FUNCTION "FC_SPL_PLC1" : VOID
TITLE =
//$Revision: 1.12 $
//$Date: 2007/10/19 12:45:04CEST $
//$Author: hgc $
//
//
//
//PLC-SPL Baustein für Solutionline DMx55-125x2
//
//Unterteilt in zwei Sicherheitsbereiche:
//1. Bereich 1         (Arbeitsraumachsen / Palettenwechslerachse / Mgazinachsen)
//bestehend aus Achse:    X Y Z B C SPI              PW             MAG1/MAG2 GR
//
//2. Bereich 2         (Palettenspeicherachsen / Palettenwechslerachse)
//bestehend aus Achse:     DREHST/TRANSP/HUB              PW
//
AUTHOR : GehAB
FAMILY : SPL
VERSION : 3.0


VAR_TEMP
  TX_ABNAHME_TEST_SBH_AKT : BOOL ;
END_VAR
BEGIN
NETWORK
TITLE =PLC-->NC: Vorbesetzungen
// Reissleine
      SET   ;
      =     "DB_SPL".IPLC_NEG_NOT_HALT;
      =     "DB_SIEM_NCK".A_Disabl_Out1;
      =     "DB_SIEM_NCK".A_OvMask_Out1;
      =     "DB_SIEM_NCK".A_Set_Out1;
      CLR   ;
      =     "DB_SIEM_NCK".A_Disabl_Out2;
      =     "DB_SIEM_NCK".A_Disabl_Out3;
      SET   ;
      =     "DB_SIEM_NCK".A_OvMask_Out2;
      =     "DB_SIEM_NCK".A_OvMask_Out3;
NETWORK
TITLE =PLC-->NC: Safety Abnahme läuft
// kein NOT-AUS auslösen und nicht SBH/SG abwählen bei Fehler SG/SGH
      U     "DB_PLC_MD_DB20".UDHex._05_BIT2_SAFTY_ABNAHME;
      =     "DB_SPL".IPLC_Abnahme;
NETWORK
TITLE =PLC-->NC: Zwangsdynamisierung laeuft
//kein Not-AUS auslösen
      U(    ;
      U(    ;
      O     "DB_SAFE_ZD".Seco_Test.Test_HW_laueft;
      O     "DB_SAFE_ZD".Seco_Test.Test_ABSP_laeuft;
      O     "DB_SAFE_ZD".Seco_Test.Test_extStop_laeuft;
      O     "DB_SAFE_ZD".Seco_Test.Test_Bremse_laeuft;
      O     ;
      U(    ;
      O     "DB_SAFE_ZD".Seco_Test.BER2_Test_HW_laueft;
      O     "DB_SAFE_ZD".Seco_Test.BER2_Test_ABSP_laeuft;
      O     "DB_SAFE_ZD".Seco_Test.BER2_Test_extStop_laeuft;
      O     "DB_SAFE_ZD".Seco_Test.BER2_Test_Bremse_laeuft;
      )     ;
      UN    "m_inbetrieb_logisch_1";
      )     ;
      S     "DB_SAFE_ALLG1".M_IMP_Test_HW_laueft;
      U(    ;
      U(    ;
      O     "DB_SAFE_ZD".Seco_Test.Test_extStop_laeuft;
      O     ;
      U     "DB_SAFE_ZD".Seco_Test.BER2_Test_extStop_laeuft;
      UN    "m_inbetrieb_logisch_1";
      )     ;
      FN    "DB_SAFE_ALLG1".M_FP_Test_HW_laueft;
      O     "M_Ruecksetze_Fehler";
      )     ;
      R     "DB_SAFE_ALLG1".M_IMP_Test_HW_laueft;
      U     "DB_SAFE_ALLG1".M_IMP_Test_HW_laueft;
      )     ;
      L     S5T#1S;
      SA    "T_SA_HW_Test_laeuft";
      NOP   0;
      NOP   0;
      NOP   0;
      U     "T_SA_HW_Test_laeuft";
      =     "DB_SPL".IPLC_ZD_GR1_RUN;
NETWORK
TITLE =PLC-->NC: ARBEITSRAUM: SBH Anforderung durch Anwahl Entriegeln
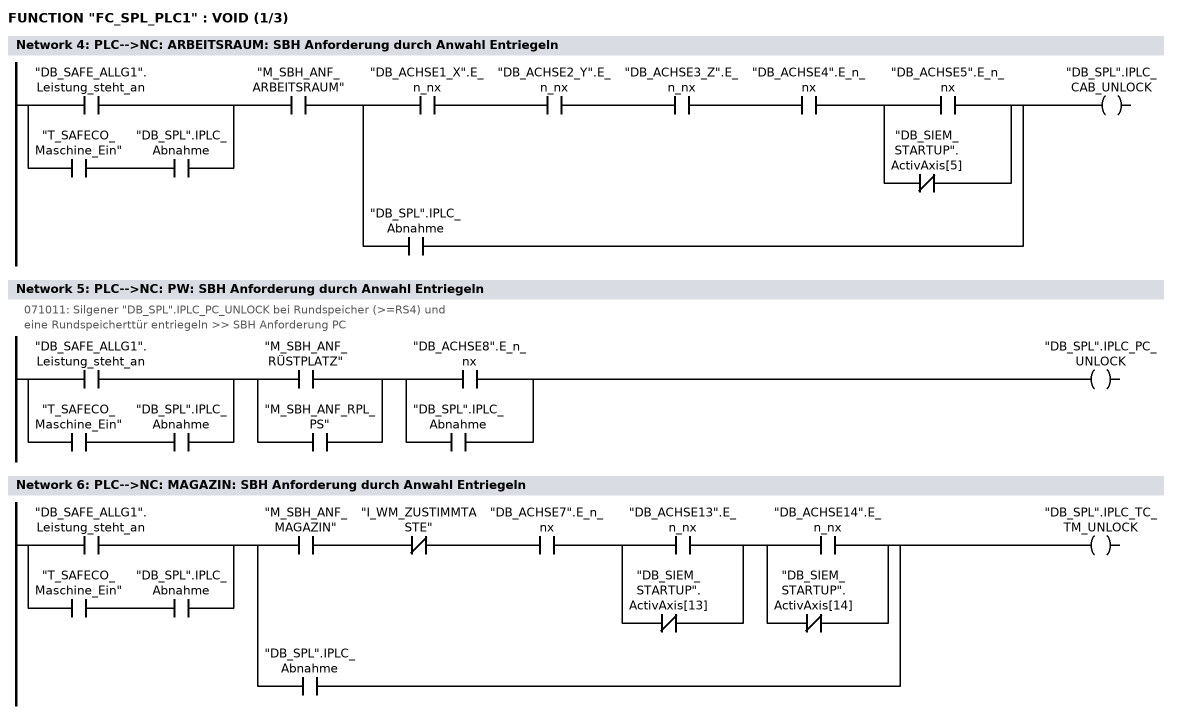

      U(    ;
      O     "DB_SAFE_ALLG1".Leistung_steht_an;
      O     ;
      U     "T_SAFECO_Maschine_Ein";
      U     "DB_SPL".IPLC_Abnahme;
      )     ;
      U     "M_SBH_ANF_ARBEITSRAUM";
      U(    ;
      U     "DB_ACHSE1_X".E_n_nx;
      U     "DB_ACHSE2_Y".E_n_nx;
      U     "DB_ACHSE3_Z".E_n_nx;
      U     "DB_ACHSE4".E_n_nx;
      U(    ;
      O     "DB_ACHSE5".E_n_nx;
      ON    "DB_SIEM_STARTUP".ActivAxis[5];
      )     ;
      O     "DB_SPL".IPLC_Abnahme;
      )     ;
      =     "DB_SPL".IPLC_CAB_UNLOCK;
NETWORK
TITLE =PLC-->NC: PW: SBH Anforderung durch Anwahl Entriegeln
//071011: Silgener "DB_SPL".IPLC_PC_UNLOCK bei Rundspeicher (>=RS4) und
//eine Rundspeicherttür entriegeln >> SBH Anforderung PC
      U(    ;
      O     "DB_SAFE_ALLG1".Leistung_steht_an;
      O     ;
      U     "T_SAFECO_Maschine_Ein";
      U     "DB_SPL".IPLC_Abnahme;
      )     ;
      U(    ;
      O     "M_SBH_ANF_RÜSTPLATZ";
      O     "M_SBH_ANF_RPL_PS";
      )     ;
      U(    ;
      O     "DB_ACHSE8".E_n_nx;
      O     "DB_SPL".IPLC_Abnahme;
      )     ;
      =     "DB_SPL".IPLC_PC_UNLOCK;
NETWORK
TITLE =PLC-->NC: MAGAZIN: SBH Anforderung durch Anwahl Entriegeln

      U(    ;
      O     "DB_SAFE_ALLG1".Leistung_steht_an;
      O     ;
      U     "T_SAFECO_Maschine_Ein";
      U     "DB_SPL".IPLC_Abnahme;
      )     ;
      U(    ;
      U     "M_SBH_ANF_MAGAZIN";
      UN    "I_WM_ZUSTIMMTASTE";
      U     "DB_ACHSE7".E_n_nx;
      U(    ;
      O     "DB_ACHSE13".E_n_nx;
      ON    "DB_SIEM_STARTUP".ActivAxis[13];
      )     ;
      U(    ;
      O     "DB_ACHSE14".E_n_nx;
      ON    "DB_SIEM_STARTUP".ActivAxis[14];
      )     ;
      O     "DB_SPL".IPLC_Abnahme;
      )     ;
      =     "DB_SPL".IPLC_TC_TM_UNLOCK;

NETWORK
TITLE =Sichere Eingänge auf Merker abbilden
//"DB_SPL".ISX_TM_DRIVES_EN_CNC  entspricht dem Eingang "IX_TC_ENABLE" (beide
//Signale durch PNOZ Multi gleichgeschaltet)
//
//"DB_SPL".ISX_PC_DRIVES_EN_CNC entspricht dem Eingang "IX_PC_ENABLE" (beide
//Signale durch PNOZ Multi gleichgeschaltet)
//
//Die Eingänge "IX_TC_ENABLE" und "IX_PC_ENABLE" werden im Rangierer auf
//Dummymerker gelegt. In der PLC wird nur das Profisafeeingangssignal abgefragt.
//
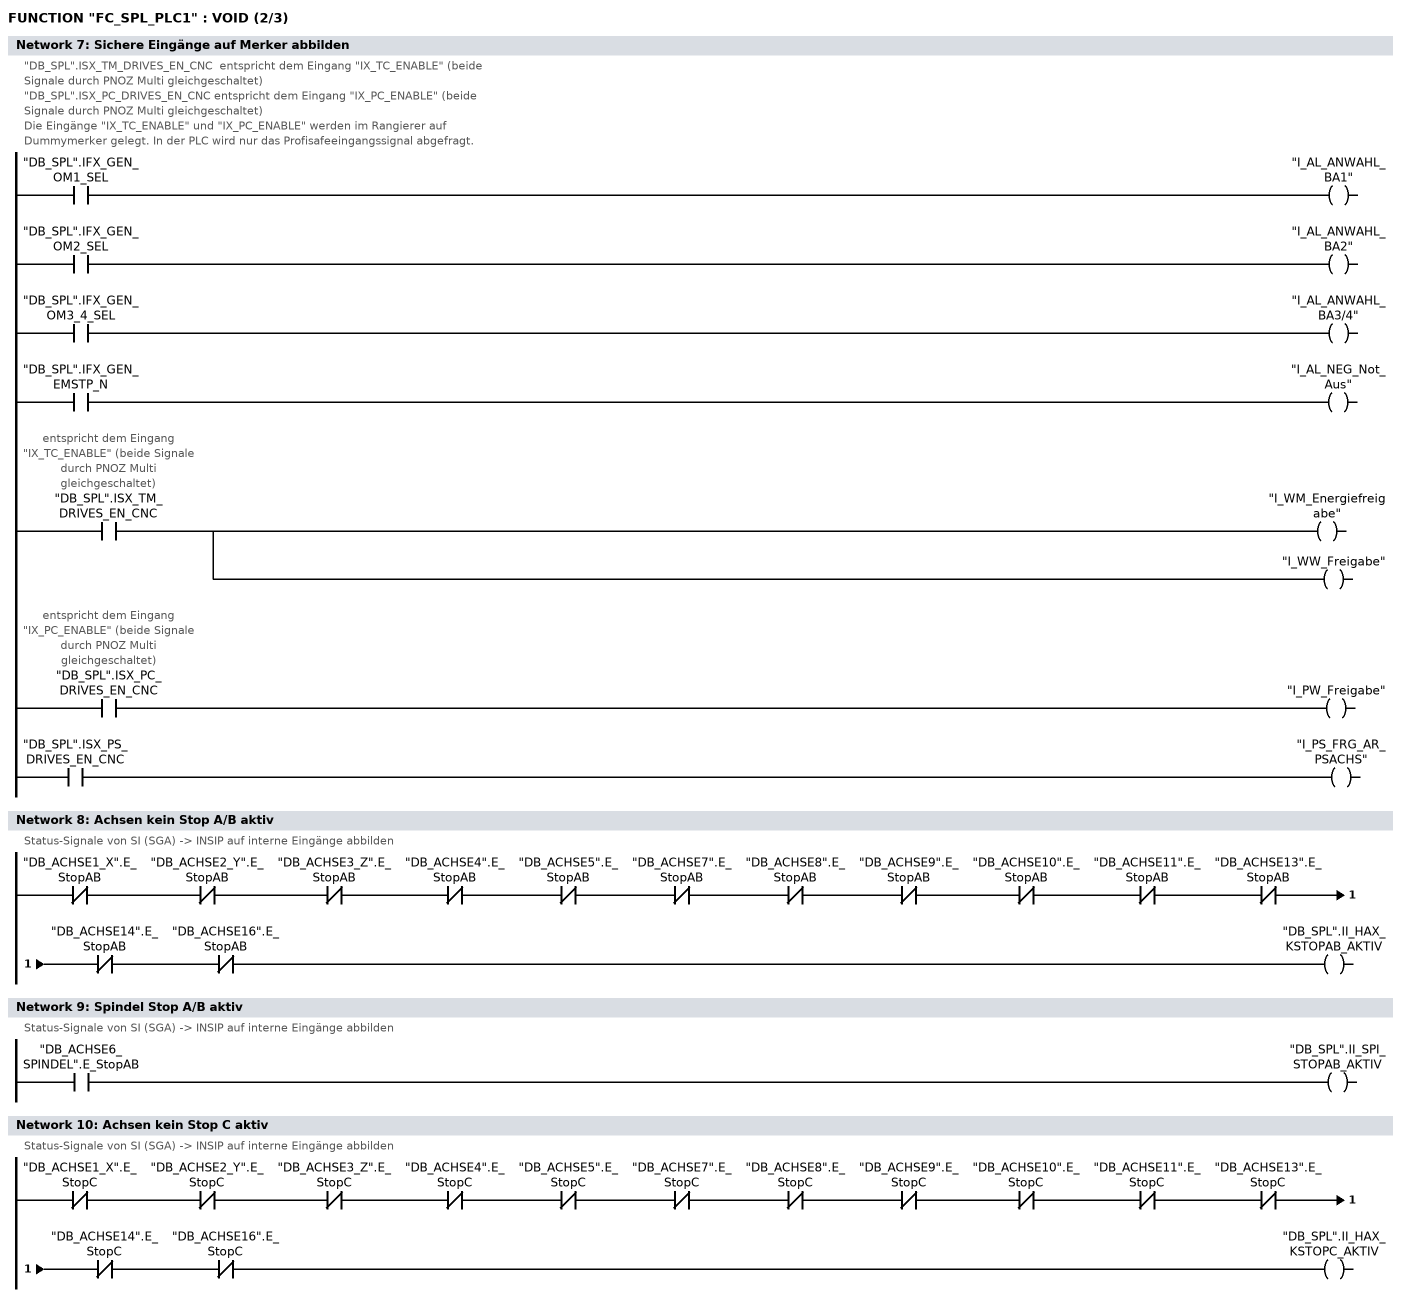
      U     "DB_SPL".IFX_GEN_OM1_SEL;
      =     "I_AL_ANWAHL_BA1";

      U     "DB_SPL".IFX_GEN_OM2_SEL;
      =     "I_AL_ANWAHL_BA2";

      U     "DB_SPL".IFX_GEN_OM3_4_SEL;
      =     "I_AL_ANWAHL_BA3/4";

      U     "DB_SPL".IFX_GEN_EMSTP_N;
      =     "I_AL_NEG_Not_Aus";

      U     "DB_SPL".ISX_TM_DRIVES_EN_CNC; // entspricht dem Eingang "IX_TC_ENABLE" (beide Signale durch PNOZ Multi gleichgeschaltet)
      =     "I_WM_Energiefreigabe";
      =     "I_WW_Freigabe";

      U     "DB_SPL".ISX_PC_DRIVES_EN_CNC; // entspricht dem Eingang "IX_PC_ENABLE" (beide Signale durch PNOZ Multi gleichgeschaltet)
      =     "I_PW_Freigabe";

      U     "DB_SPL".ISX_PS_DRIVES_EN_CNC;
      =     "I_PS_FRG_AR_PSACHS";
NETWORK
TITLE =Achsen kein Stop A/B aktiv
//Status-Signale von SI (SGA) -> INSIP auf interne Eingänge abbilden
      UN    "DB_ACHSE1_X".E_StopAB;
      UN    "DB_ACHSE2_Y".E_StopAB;
      UN    "DB_ACHSE3_Z".E_StopAB;
      UN    "DB_ACHSE4".E_StopAB;
      UN    "DB_ACHSE5".E_StopAB;
      UN    "DB_ACHSE7".E_StopAB;
      UN    "DB_ACHSE8".E_StopAB;
      UN    "DB_ACHSE9".E_StopAB;
      UN    "DB_ACHSE10".E_StopAB;
      UN    "DB_ACHSE11".E_StopAB;
      UN    "DB_ACHSE13".E_StopAB;
      UN    "DB_ACHSE14".E_StopAB;
      UN    "DB_ACHSE16".E_StopAB;
      =     "DB_SPL".II_HAX_KSTOPAB_AKTIV;
NETWORK
TITLE =Spindel Stop A/B aktiv
//Status-Signale von SI (SGA) -> INSIP auf interne Eingänge abbilden
      U     "DB_ACHSE6_SPINDEL".E_StopAB;
      =     "DB_SPL".II_SPI_STOPAB_AKTIV;
NETWORK
TITLE =Achsen kein Stop C aktiv
//Status-Signale von SI (SGA) -> INSIP auf interne Eingänge abbilden
      UN    "DB_ACHSE1_X".E_StopC;
      UN    "DB_ACHSE2_Y".E_StopC;
      UN    "DB_ACHSE3_Z".E_StopC;
      UN    "DB_ACHSE4".E_StopC;
      UN    "DB_ACHSE5".E_StopC;
      UN    "DB_ACHSE7".E_StopC;
      UN    "DB_ACHSE8".E_StopC;
      UN    "DB_ACHSE9".E_StopC;
      UN    "DB_ACHSE10".E_StopC;
      UN    "DB_ACHSE11".E_StopC;
      UN    "DB_ACHSE13".E_StopC;
      UN    "DB_ACHSE14".E_StopC;
      UN    "DB_ACHSE16".E_StopC;
      =     "DB_SPL".II_HAX_KSTOPC_AKTIV;
NETWORK
TITLE =Spindel Stop C aktiv
//Status-Signale von SI (SGA) -> INSIP auf interne Eingänge abbilden
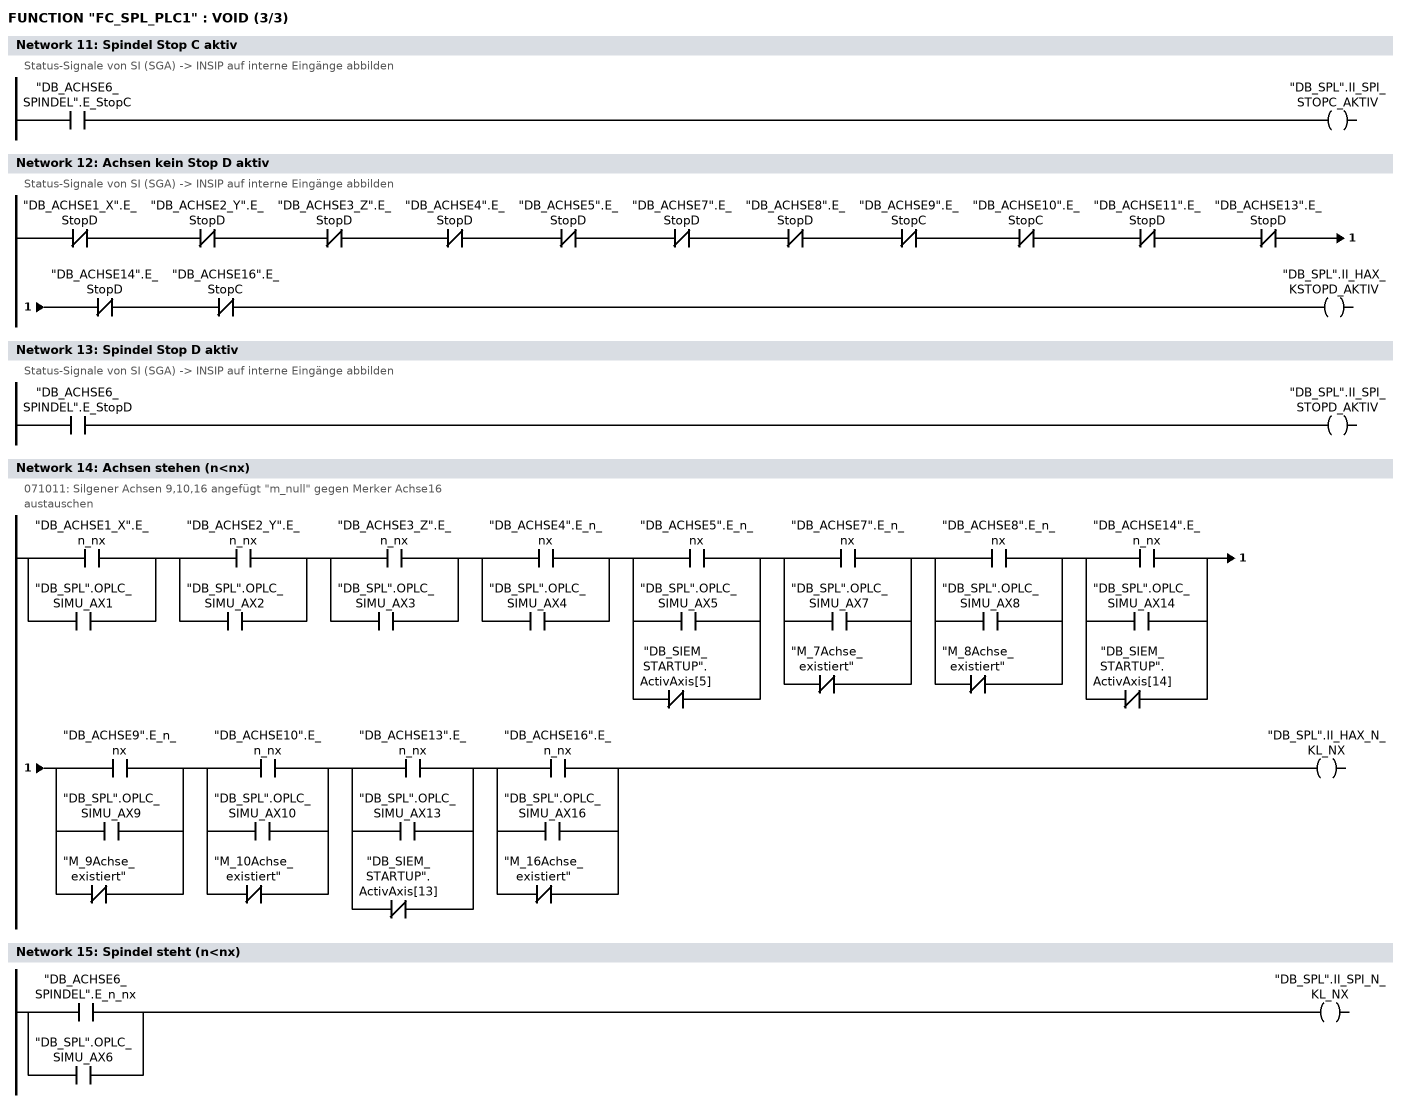
      U     "DB_ACHSE6_SPINDEL".E_StopC;
      =     "DB_SPL".II_SPI_STOPC_AKTIV;
NETWORK
TITLE =Achsen kein Stop D aktiv
//Status-Signale von SI (SGA) -> INSIP auf interne Eingänge abbilden
      UN    "DB_ACHSE1_X".E_StopD;
      UN    "DB_ACHSE2_Y".E_StopD;
      UN    "DB_ACHSE3_Z".E_StopD;
      UN    "DB_ACHSE4".E_StopD;
      UN    "DB_ACHSE5".E_StopD;
      UN    "DB_ACHSE7".E_StopD;
      UN    "DB_ACHSE8".E_StopD;
      UN    "DB_ACHSE9".E_StopC;
      UN    "DB_ACHSE10".E_StopC;
      UN    "DB_ACHSE11".E_StopD;
      UN    "DB_ACHSE13".E_StopD;
      UN    "DB_ACHSE14".E_StopD;
      UN    "DB_ACHSE16".E_StopC;
      =     "DB_SPL".II_HAX_KSTOPD_AKTIV;
NETWORK
TITLE =Spindel Stop D aktiv
//Status-Signale von SI (SGA) -> INSIP auf interne Eingänge abbilden
      U     "DB_ACHSE6_SPINDEL".E_StopD;
      =     "DB_SPL".II_SPI_STOPD_AKTIV;
NETWORK
TITLE =Achsen stehen (n<nx)
//071011: Silgener Achsen 9,10,16 angefügt "m_null" gegen Merker Achse16
//austauschen
      U(    ;
      O     "DB_ACHSE1_X".E_n_nx;
      O     "DB_SPL".OPLC_SIMU_AX1;
      )     ;
      U(    ;
      O     "DB_ACHSE2_Y".E_n_nx;
      O     "DB_SPL".OPLC_SIMU_AX2;
      )     ;
      U(    ;
      O     "DB_ACHSE3_Z".E_n_nx;
      O     "DB_SPL".OPLC_SIMU_AX3;
      )     ;
      U(    ;
      O     "DB_ACHSE4".E_n_nx;
      O     "DB_SPL".OPLC_SIMU_AX4;
      )     ;
      U(    ;
      O     "DB_ACHSE5".E_n_nx;
      O     "DB_SPL".OPLC_SIMU_AX5;
      ON    "DB_SIEM_STARTUP".ActivAxis[5];
      )     ;
      U(    ;
      O     "DB_ACHSE7".E_n_nx;
      O     "DB_SPL".OPLC_SIMU_AX7;
      ON    "M_7Achse_existiert";
      )     ;
      U(    ;
      O     "DB_ACHSE8".E_n_nx;
      O     "DB_SPL".OPLC_SIMU_AX8;
      ON    "M_8Achse_existiert";
      )     ;
      U(    ;
      O     "DB_ACHSE14".E_n_nx;
      O     "DB_SPL".OPLC_SIMU_AX14;
      ON    "DB_SIEM_STARTUP".ActivAxis[14];
      )     ;
      U(    ;
      O     "DB_ACHSE9".E_n_nx;
      O     "DB_SPL".OPLC_SIMU_AX9;
      ON    "M_9Achse_existiert";
      )     ;
      U(    ;
      O     "DB_ACHSE10".E_n_nx;
      O     "DB_SPL".OPLC_SIMU_AX10;
      ON    "M_10Achse_existiert";
      )     ;
      U(    ;
      O     "DB_ACHSE13".E_n_nx;
      O     "DB_SPL".OPLC_SIMU_AX13;
      ON    "DB_SIEM_STARTUP".ActivAxis[13];
      )     ;
      U(    ;
      O     "DB_ACHSE16".E_n_nx;
      O     "DB_SPL".OPLC_SIMU_AX16;
      ON    "M_16Achse_existiert";
      )     ;
      =     "DB_SPL".II_HAX_N_KL_NX;
NETWORK
TITLE =Spindel steht (n<nx)

      O     "DB_ACHSE6_SPINDEL".E_n_nx;
      O     "DB_SPL".OPLC_SIMU_AX6;
      =     "DB_SPL".II_SPI_N_KL_NX;
NETWORK
TITLE =SPL-Logik INSEP/INSIP -> OUTSIP abbilden: Schutzbereich Maschin
//vgl. SAFE.SPF
//$A_MARKERSIP[1]...$A_MARKERSIP[64] : DB18.DBX70.0 ... DB18.DBX77.7
//$A_OUTSIP[1]......$A_OUTSIP[64]    : DB18.DBX62.0 ... DB18.DBX69.7
//
//--- Anforderung ST öffnen
//--- PLC- Eingaenge --> an NC
//--- NOT-HALT
// MK_NEG_NOT_HALT = (IX_AL_Drehzahl_Max==1) OR (IX_AL_BA2==1) OR (IX_AL_BA34==1)
      NOP   0;
// merker werden in NCK-SPL um 20 ms gegenüber dem Eingang verzögert
// weil das PNOZ-multi die Signale mit 200 us taktet

      U     "DB_SPL".IFX_GEN_OM1_SEL;
      =     "DB_SPL".MX_HAX_VERZ;

      U     "DB_SPL".IFX_GEN_OM2_SEL;
      =     "DB_SPL".MARKERSIP12;

      U     "DB_SPL".IFX_GEN_OM3_4_SEL;
      =     "DB_SPL".MARKERSIP13;

      U     "DB_SPL".IFX_GEN_EMSTP_N;
      =     "DB_SPL".MARKERSIP14;

//-------------------------------------------------------------------

      O     "DB_SPL".IFX_GEN_OM1_SEL;
      O     "DB_SPL".IFX_GEN_OM2_SEL;
      O     "DB_SPL".IFX_GEN_OM3_4_SEL;
      U     "DB_SPL".IFX_GEN_EMSTP_N;
      U     "DB_SPL".IPLC_NEG_NOT_HALT;
      =     "DB_SPL".MK_NEG_NOT_HALT;

      U     "DB_SPL".IFX_GEN_EMSTP_N;
      =     "DB_SPL".MK_NEG_NOT_TAST;

// SBH-Abwahl------------------------------------------------------------
//N1020 IDS=58 DO OI_SBH_ABW_HAX = MK_NEG_NOT_HALT OI_SBH_ABW_SPI = MK_NEG_NOT_HALT
//N1025 IDS=59 DO OI_SBH_ABW_TC = MK_NEG_NOT_HALT AND ISX_TC_DRIVES_EN_CNC
//N1030 IDS=60 DO OI_SBH_ABW_TM = MK_NEG_NOT_HALT AND ISX_TM_DRIVES_EN_CNC
//N1035 IDS=61 DO OI_SBH_ABW_PW = MK_NEG_NOT_HALT AND ISX_PC_DRIVES_EN_CNC

      U     "I_AL_ANWAHL_BA3/4";
      O     "I_AL_ANWAHL_BA2";
      O(    ;
      U     "DB_SPL".MK_NEG_NOT_HALT;
      UN    "DB_SPL".IPLC_CAB_UNLOCK;
      )     ;
      =     "DB_SPL".OI_SBH_ABW_HAX;
      =     "DB_SPL".OI_SBH_ABW_SPI;


      U     "DB_SPL".MK_NEG_NOT_HALT;
      U     "DB_SPL".ISX_TC_DRIVES_EN_CNC;
      UN    "DB_SPL".IPLC_TC_TM_UNLOCK;
      UN    "DB_SPL".IPLC_CAB_UNLOCK;
      UN    "I_AL_ANWAHL_BA3/4";
      UN    "I_AL_ANWAHL_BA2";
      =     "DB_SPL".OI_SBH_ABW_TC;

      UN    "DB_SPL".IPLC_TC_TM_UNLOCK;
      =     "DB_SPL".OI_SBH_ABW_TM;

      U     "DB_SPL".MK_NEG_NOT_HALT;
      U     "DB_SPL".ISX_PC_DRIVES_EN_CNC;
      UN    "DB_SPL".IPLC_PC_UNLOCK;
      =     "DB_SPL".OI_SBH_ABW_PC;



//-----------------------------------------------------------------------


// SBH/SG-Abwahl---------------------------------------------------------
//N1030 IDS=53 DO OI_SBH_SG_ABW_HAX = MK_NEG_NOT_HALT OI_SBH_SG_ABW_SPI = (NOT MK_NEG_NOT_HALT) OR II_SPI_STOPAB_AKTIV

      ON    "DB_SPL".MK_NEG_NOT_TAST;
      O(    ;
      UN    "DB_SPL".II_HAX_KSTOPAB_AKTIV;
      UN    "DB_SPL".IPLC_Abnahme;
      )     ;
      =     "DB_SPL".OI_SBH_SG_ABW_HAX;

      O     "DB_SPL".II_SPI_STOPAB_AKTIV;
      ON    "DB_SPL".MK_NEG_NOT_HALT;
//  O     "SPL".IPLC_Abnahme
      =     "DB_SPL".OI_SBH_SG_ABW_SPI;

//-----------------------------------------------------------------------


// SG-Auswahl------------------------------------------------------------
//N1040 IDS=53 DO OI_SG_AUSW_24_HAX = MIX_AL_BA2 AND (NOT MIX_AL_BA34) AND (NOT MIX_AL_Drehzahl_Max)
//N1045 IDS=83 DO OI_SG_AUSW_24_MAGAX = OI_SG_AUSW_24_HAX AND IPLC_Abnahme
//N1050 IDS=54 DO OI_SG_AUSW_34_HAX = (MIX_AL_BA34 AND (NOT MIX_AL_Drehzahl_Max)) OR IPLC_TEST_BA4
//N1055 IDS=85 DO OI_SG_AUSW_34_MAGAX = OI_SG_AUSW_34_HAX AND IPLC_Abnahme

      U     "DB_SPL".IFX_GEN_OM2_SEL; // BA 2
      UN    "DB_SPL".IFX_GEN_OM3_4_SEL;
      UN    "DB_SPL".IFX_GEN_OM1_SEL;
      =     "DB_SPL".OI_SG_AUSW_24_HAX;

      U     "DB_SPL".OI_SG_AUSW_24_HAX; // BA 2 währende SI-Abnahme
      U     "DB_SPL".IPLC_Abnahme;
      =     "DB_SPL".OI_SG_AUSW_24_MAGAX;



      U     "DB_SPL".IFX_GEN_OM3_4_SEL; // BA 34
      UN    "DB_SPL".IFX_GEN_OM1_SEL;
      O     "DB_SPL".IPLC_Test_BA4;
      =     "DB_SPL".OI_SG_AUSW_34_HAX;

      U     "DB_SPL".OI_SG_AUSW_34_HAX; // BA 34 währende SI-Abnahme
      U     "DB_SPL".IPLC_Abnahme;
      =     "DB_SPL".OI_SG_AUSW_34_MAGAX;

//-----------------------------------------------------------------------


//--- Externer Stopp A- Abwahl : Spindel
//--- Wenn keine Betriebsart mehr aktiv ist dann Spindel stoppen

      U     "DB_SPL".MK_NEG_NOT_HALT; // Not-Halt gesamt
      L     S5T#5S;
      SA    "T_SAFECO_STOPA_SPI";
      U     "T_SAFECO_STOPA_SPI";
      =     "DB_SPL".MK_STOPA_NH_SPI; // HM STOP A von Not-Halt Hauptachsen

      U     "DB_SPL".OI_SBH_ABW_HAX; // Abwahl STOP A Hauptachsen
      S     "DB_SPL".MK_KSTOPA_NX_SPI;
      U     "DB_SPL".II_SPI_N_KL_NX;
      R     "DB_SPL".MK_KSTOPA_NX_SPI;

      U     "DB_SPL".MK_STOPA_NH_SPI; // HM STOP A von Not-Halt Hauptachsen
      UN    "DB_SAFE_ZD".GR1_ZD.req_stopa_plc; // Zwangsdyn. STOP A (PLC)
      U(    ;
      O     "DB_SPL".OI_SBH_ABW_HAX;
      O     "DB_SPL".MK_KSTOPA_NX_SPI; // HM STOP A von Not-Halt
      )     ;
      =     "DB_SPL".OI_STOPA_ABW_SPI; // Abwahl STOP A

//--- Externer Stopp A- Abwahl : Hauptachsen

      L     "DB_PLC_MD_DB20".UDInt._005_ANWAHL_SONDER_SPDL; //Option Drehbetrieb wenn Hirthverzahnung
      L     2;
      ==I   ;
      SPBN  n4a;
      U     "DB_SPL".MK_NEG_NOT_TAST; // Not-Halt gesamt
      L     S5T#8S;
      SA    "T_NH_STOPA_AX";
      U     "T_NH_STOPA_AX";
      =     "DB_SPL".MK_STOPA_NH_AX; // HM STOP A von Not-Halt Hauptachsen
      SPA   n4b;

n4a:  U     "DB_SPL".MK_NEG_NOT_TAST; // Not-Halt gesamt
      L     S5T#1S;
      SA    "T_NH_STOPA_AX";
      U     "T_NH_STOPA_AX";
      =     "DB_SPL".MK_STOPA_NH_AX; // HM STOP A von Not-Halt Hauptachsen

n4b:  U     "DB_SPL".MK_STOPA_NH_AX; // HM STOP A von Not-Halt Hauptachsen
      UN    "DB_SAFE_ZD".GR1_ZD.req_stopa_plc; // Zwangsdyn. STOP A (PLC)
      =     "DB_SPL".OI_STOPA_ABW_HAX; // Abwahl STOP A

//--- Externer Stopp D- Abwahl : Hauptachsen

      UN    "DB_SAFE_ZD".GR1_ZD.req_stopd_plc; // Zwangsdyn. STOP D (PLC)
      =     "DB_SPL".OI_STOPD_ABW_HAX;

//--- Externer Stopp D- Abwahl : Palettenwechslerachse

      O(    ;
      U     "DB_SPL".OI_STOPD_ABW_HAX;
      U     "DB_SPL".MK_NEG_NOT_TAST;
      UN    "DB_SPL".IPLC_ZD_GR1_RUN;
      )     ;
      O(    ;
      U     "DB_SPL".OI_STOPC_ABW_HAX;
      U     "DB_SPL".IPLC_ZD_GR1_RUN;
      )     ;
      =     "DB_SPL".OI_STOPD_ABW_PC;



//--- Externer Stopp C - Abwahl : Hauptachsen

      U     "DB_SPL".MK_NEG_NOT_TAST;
      UN    "DB_SAFE_ZD".GR1_ZD.req_stopc_plc; // Zwangsdyn. STOP C (PLC)
      =     "DB_SPL".OI_STOPC_ABW_HAX;

//--- Externer Stopp C- Abwahl : Palettenwechslerachse

      UN    "DB_SPL".IPLC_ZD_GR1_RUN;
      O(    ;
      U     "DB_SPL".OI_STOPC_ABW_HAX;
      U     "DB_SPL".IPLC_ZD_GR1_RUN;
      )     ;
      =     "DB_SPL".OI_STOPC_ABW_PC;





// Zwangsdynamisierung
      U     "DB_SPL".IPLC_ZD_Gr1_EXT;
      =     "DB_SPL".OI_ZD_Gr1_EXT;

//--- OX_AL_NEG_NOT_HALT-------------------------------------------------
// Bei Zwangsdynamisierung wird kein NOT-HALT ausgegeben

      ON    "DB_SPL".II_HAX_KSTOPC_AKTIV;
      O     "DB_SPL".II_SPI_STOPC_AKTIV;
      ON    "DB_SPL".II_HAX_KSTOPD_AKTIV;
      O     "DB_SPL".II_SPI_STOPD_AKTIV;
      ON    "DB_SPL".II_HAX_KSTOPAB_AKTIV;
      L     S5T#1S;
      SV    "T_DREHZAHL_OK";

      U     "T_DREHZAHL_OK";
      UN    "DB_SPL".IPLC_ZD_GR1_RUN;
      UN    "DB_SPL".IPLC_Abnahme;
      =     "DB_SPL".MX_AL_DREHZAHL_OK;

//-----------------------------------------------------------------------

      UN    "DB_SPL".MX_AL_DREHZAHL_OK;
      =     "DB_SPL".OFX_GEN_EMSTP_N;

// OX_AL_HAX_stehen------------------------------------------------------
// Takt für das Signal alle 300 ms
// Ergebnis an NC mitteilen
// in NC Takt-Merker überwachen

      UN    "T_HAX_Stehen";
      =     "DB_SPL".IPLC_RES_13; //IPLC_Takt
      L     S5T#300MS;
      SV    "T_HAX_Stehen";

      UN    "DB_SPL".IPLC_RES_13;
      SPB   xx1;
      U     "DB_SPL".II_HAX_N_KL_NX;
      U     "DB_SPL".II_SPI_N_KL_NX;
      =     "DB_SPL".IPLC_Stehen; // an NC

      U     "DB_SPL".IPLC_Stehen; // von PLC
      U     "DB_SPL".OPLC_Stehen; // von NC aus letztem Takt
      =     "DB_SPL".OFX_GEN_STOP_MONITOR;
//-----------------------------------------------------------------------

xx1:  NOP   0;

NETWORK
TITLE = OX_AL_NEG_NOT_HALT
//Ext.Ausgänge (OUTSEP) an Peripherie ausgeben
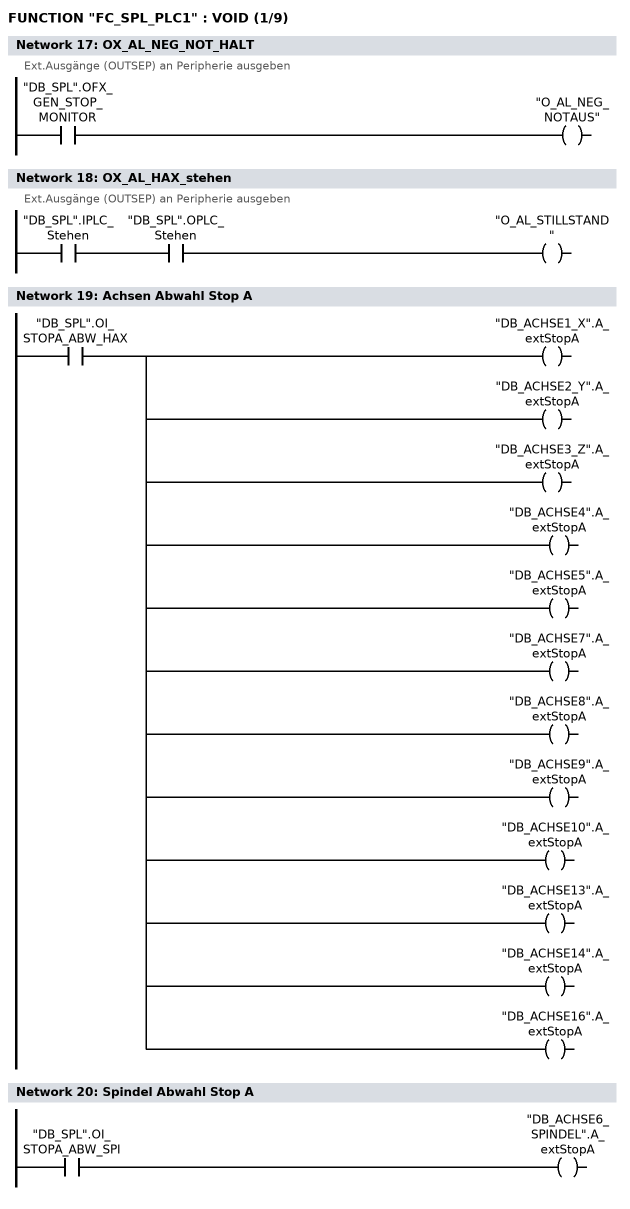
      U     "DB_SPL".OFX_GEN_STOP_MONITOR;
      =     "O_AL_NEG_NOTAUS";
NETWORK
TITLE =OX_AL_HAX_stehen
//Ext.Ausgänge (OUTSEP) an Peripherie ausgeben
      U     "DB_SPL".IPLC_Stehen;
      U     "DB_SPL".OPLC_Stehen;
      =     "O_AL_STILLSTAND";
NETWORK
TITLE =Achsen Abwahl Stop A

      U     "DB_SPL".OI_STOPA_ABW_HAX;
      =     "DB_ACHSE1_X".A_extStopA;
      =     "DB_ACHSE2_Y".A_extStopA;
      =     "DB_ACHSE3_Z".A_extStopA;
      =     "DB_ACHSE4".A_extStopA;
      =     "DB_ACHSE5".A_extStopA;
      =     "DB_ACHSE7".A_extStopA;
      =     "DB_ACHSE8".A_extStopA;
      =     "DB_ACHSE9".A_extStopA;
      =     "DB_ACHSE10".A_extStopA;
      =     "DB_ACHSE13".A_extStopA;
      =     "DB_ACHSE14".A_extStopA;
      =     "DB_ACHSE16".A_extStopA;
NETWORK
TITLE =Spindel Abwahl Stop A

      U     "DB_SPL".OI_STOPA_ABW_SPI;
      =     "DB_ACHSE6_SPINDEL".A_extStopA;
NETWORK
TITLE =Achsen + Spindel Abwahl Stop C
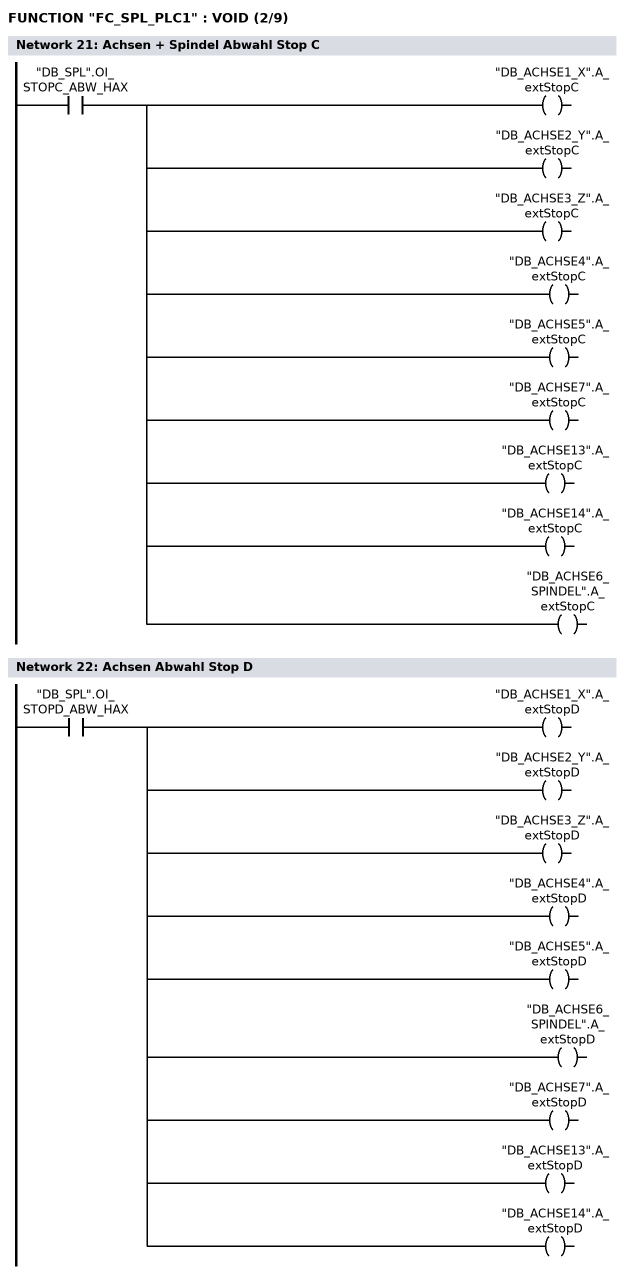

      U     "DB_SPL".OI_STOPC_ABW_HAX;
      =     "DB_ACHSE1_X".A_extStopC;
      =     "DB_ACHSE2_Y".A_extStopC;
      =     "DB_ACHSE3_Z".A_extStopC;
      =     "DB_ACHSE4".A_extStopC;
      =     "DB_ACHSE5".A_extStopC;
      =     "DB_ACHSE7".A_extStopC;
      =     "DB_ACHSE13".A_extStopC;
      =     "DB_ACHSE14".A_extStopC;
      =     "DB_ACHSE6_SPINDEL".A_extStopC;

NETWORK
TITLE =Achsen Abwahl Stop D

      U     "DB_SPL".OI_STOPD_ABW_HAX;
      =     "DB_ACHSE1_X".A_extStopD;
      =     "DB_ACHSE2_Y".A_extStopD;
      =     "DB_ACHSE3_Z".A_extStopD;
      =     "DB_ACHSE4".A_extStopD;
      =     "DB_ACHSE5".A_extStopD;
      =     "DB_ACHSE6_SPINDEL".A_extStopD;
      =     "DB_ACHSE7".A_extStopD;
      =     "DB_ACHSE13".A_extStopD;
      =     "DB_ACHSE14".A_extStopD;

NETWORK
TITLE =Achsen Abwahl Stop E
//Stop E wird gemeinsam mit Stop D abgewählt da kein ESR
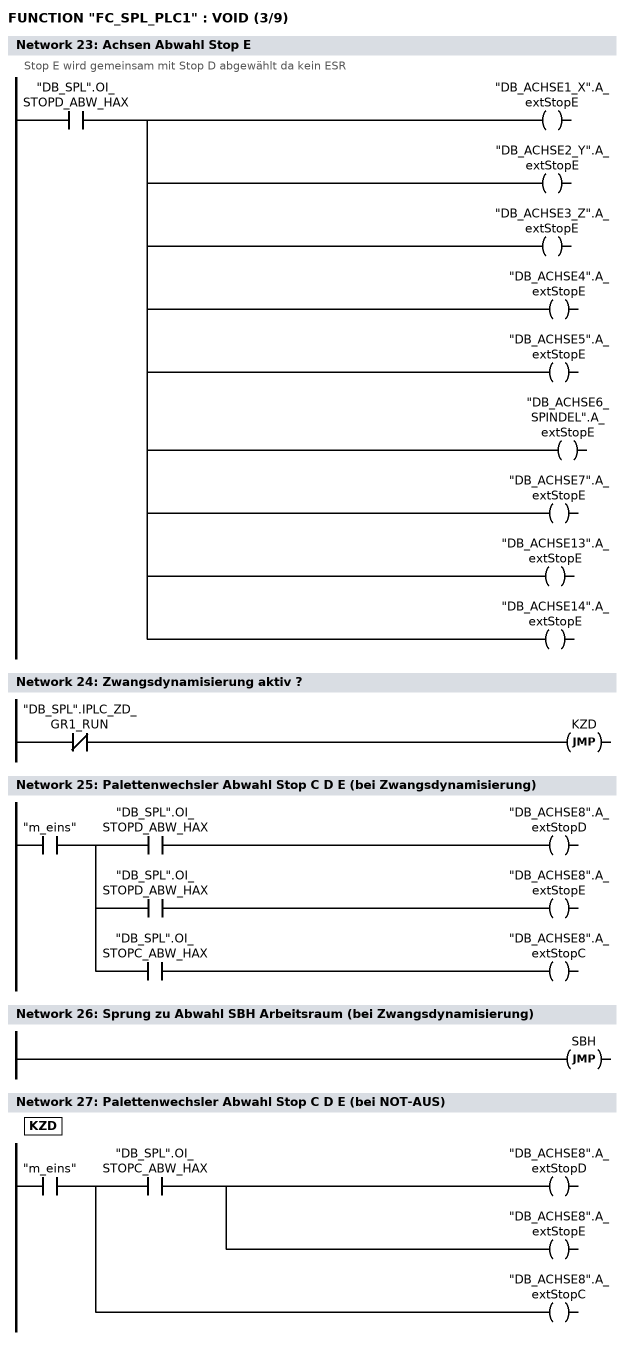
      U     "DB_SPL".OI_STOPD_ABW_HAX;
      =     "DB_ACHSE1_X".A_extStopE;
      =     "DB_ACHSE2_Y".A_extStopE;
      =     "DB_ACHSE3_Z".A_extStopE;
      =     "DB_ACHSE4".A_extStopE;
      =     "DB_ACHSE5".A_extStopE;
      =     "DB_ACHSE6_SPINDEL".A_extStopE;
      =     "DB_ACHSE7".A_extStopE;
      =     "DB_ACHSE13".A_extStopE;
      =     "DB_ACHSE14".A_extStopE;

NETWORK
TITLE =Zwangsdynamisierung aktiv ?

      UN    "DB_SPL".IPLC_ZD_GR1_RUN;
      SPB   KZD;
NETWORK
TITLE =Palettenwechsler Abwahl Stop C D E (bei Zwangsdynamisierung)

      U     "m_eins";
      =     L      1.0;
      U     L      1.0;
      U     "DB_SPL".OI_STOPD_ABW_HAX;
      =     "DB_ACHSE8".A_extStopD;
      U     L      1.0;
      U     "DB_SPL".OI_STOPD_ABW_HAX;
      =     "DB_ACHSE8".A_extStopE;
      U     L      1.0;
      U     "DB_SPL".OI_STOPC_ABW_HAX;
      =     "DB_ACHSE8".A_extStopC;
NETWORK
TITLE =Sprung zu Abwahl SBH Arbeitsraum (bei Zwangsdynamisierung)

      SPA   SBH;
NETWORK
TITLE =Palettenwechsler Abwahl Stop C D E (bei NOT-AUS)

KZD:  U     "m_eins";
      =     L      1.0;
      U     L      1.0;
      U     "DB_SPL".OI_STOPC_ABW_HAX;
      =     "DB_ACHSE8".A_extStopD;
      =     "DB_ACHSE8".A_extStopE;
      U     L      1.0;
      BLD   102;
      =     "DB_ACHSE8".A_extStopC;
NETWORK
TITLE =Abwahl SBH Arbeitsraum
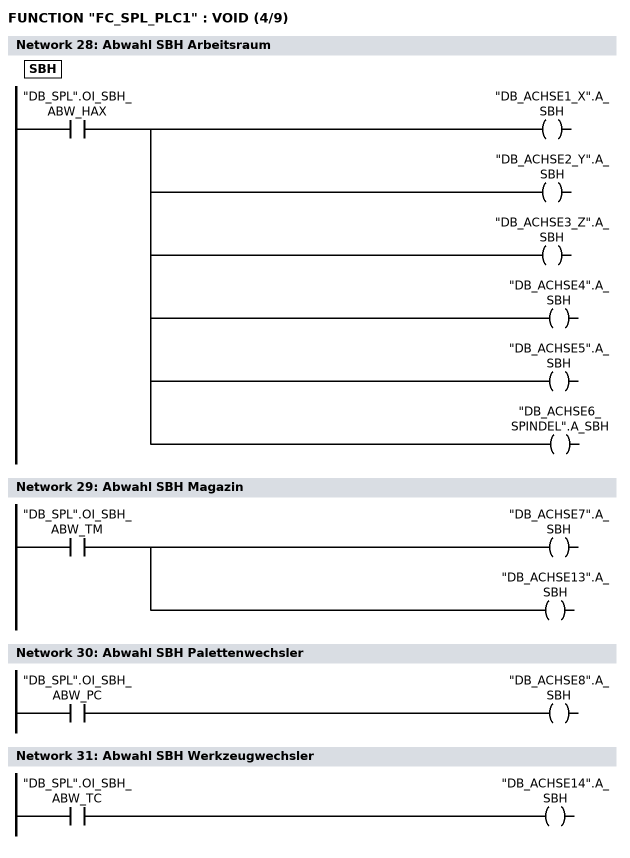

SBH:  U     "DB_SPL".OI_SBH_ABW_HAX;
      =     "DB_ACHSE1_X".A_SBH;
      =     "DB_ACHSE2_Y".A_SBH;
      =     "DB_ACHSE3_Z".A_SBH;
      =     "DB_ACHSE4".A_SBH;
      =     "DB_ACHSE5".A_SBH;
      =     "DB_ACHSE6_SPINDEL".A_SBH;
NETWORK
TITLE =Abwahl SBH Magazin

      U     "DB_SPL".OI_SBH_ABW_TM;
      =     "DB_ACHSE7".A_SBH;
      =     "DB_ACHSE13".A_SBH;
NETWORK
TITLE =Abwahl SBH Palettenwechsler

      U     "DB_SPL".OI_SBH_ABW_PC;
      =     "DB_ACHSE8".A_SBH;

NETWORK
TITLE =Abwahl SBH Werkzeugwechsler

      U     "DB_SPL".OI_SBH_ABW_TC;
      =     "DB_ACHSE14".A_SBH;
NETWORK
TITLE =Achsen SBH/SG-Abwahl
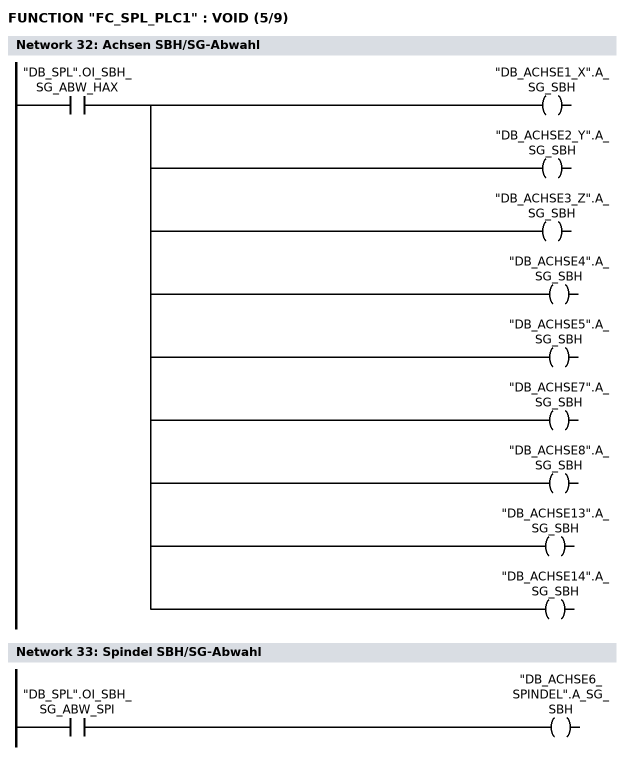

      U     "DB_SPL".OI_SBH_SG_ABW_HAX;
      =     "DB_ACHSE1_X".A_SG_SBH;
      =     "DB_ACHSE2_Y".A_SG_SBH;
      =     "DB_ACHSE3_Z".A_SG_SBH;
      =     "DB_ACHSE4".A_SG_SBH;
      =     "DB_ACHSE5".A_SG_SBH;
      =     "DB_ACHSE7".A_SG_SBH;
      =     "DB_ACHSE8".A_SG_SBH;
      =     "DB_ACHSE13".A_SG_SBH;
      =     "DB_ACHSE14".A_SG_SBH;
NETWORK
TITLE =Spindel SBH/SG-Abwahl

      U     "DB_SPL".OI_SBH_SG_ABW_SPI;
      =     "DB_ACHSE6_SPINDEL".A_SG_SBH;
NETWORK
TITLE =SG 0 -Auswahl
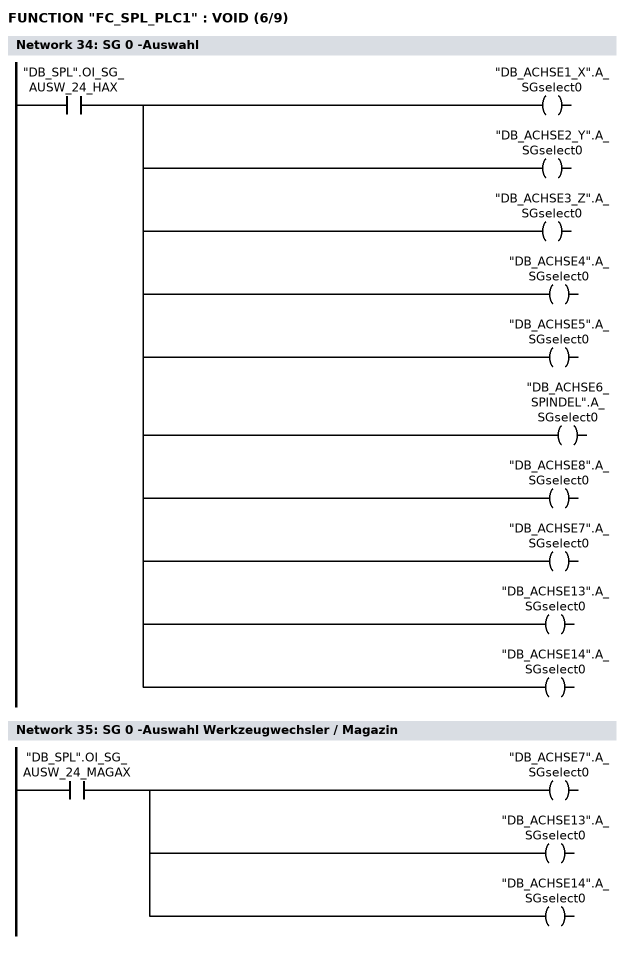

      U     "DB_SPL".OI_SG_AUSW_24_HAX;
      =     "DB_ACHSE1_X".A_SGselect0;
      =     "DB_ACHSE2_Y".A_SGselect0;
      =     "DB_ACHSE3_Z".A_SGselect0;
      =     "DB_ACHSE4".A_SGselect0;
      =     "DB_ACHSE5".A_SGselect0;
      =     "DB_ACHSE6_SPINDEL".A_SGselect0;
      =     "DB_ACHSE8".A_SGselect0;
      =     "DB_ACHSE7".A_SGselect0;
      =     "DB_ACHSE13".A_SGselect0;
      =     "DB_ACHSE14".A_SGselect0;
NETWORK
TITLE =SG 0 -Auswahl Werkzeugwechsler / Magazin

      U     "DB_SPL".OI_SG_AUSW_24_MAGAX;
      =     "DB_ACHSE7".A_SGselect0;
      =     "DB_ACHSE13".A_SGselect0;
      =     "DB_ACHSE14".A_SGselect0;
NETWORK
TITLE =SG 1 -Auswahl
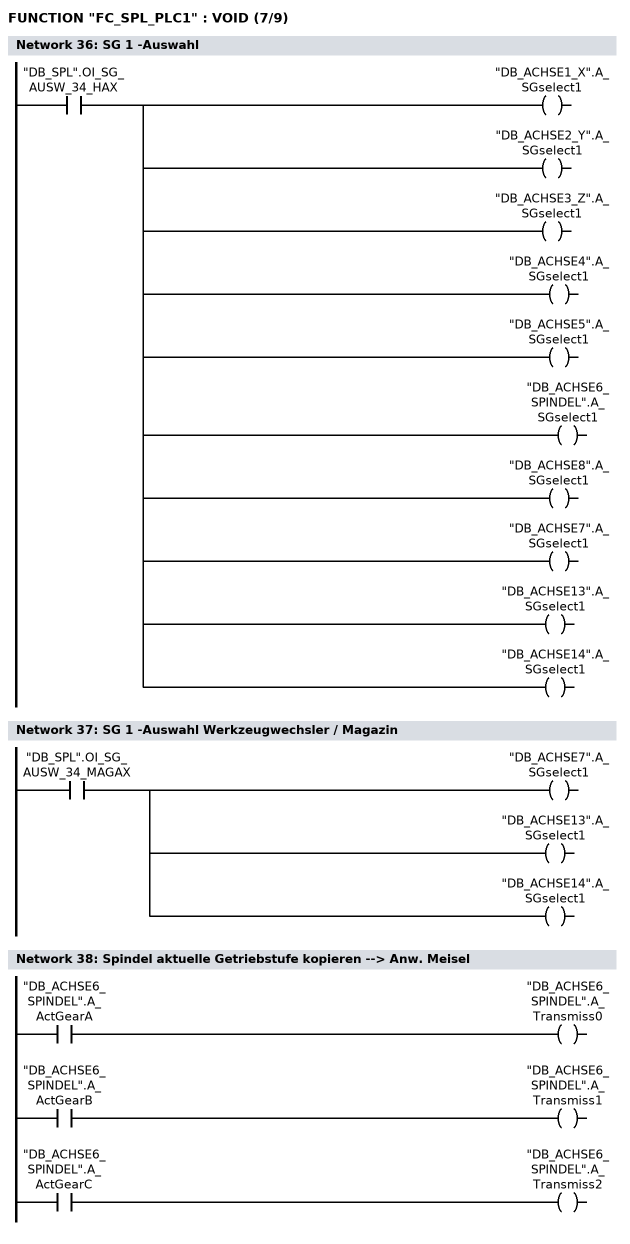

      U     "DB_SPL".OI_SG_AUSW_34_HAX;
      =     "DB_ACHSE1_X".A_SGselect1;
      =     "DB_ACHSE2_Y".A_SGselect1;
      =     "DB_ACHSE3_Z".A_SGselect1;
      =     "DB_ACHSE4".A_SGselect1;
      =     "DB_ACHSE5".A_SGselect1;
      =     "DB_ACHSE6_SPINDEL".A_SGselect1;
      =     "DB_ACHSE8".A_SGselect1;
      =     "DB_ACHSE7".A_SGselect1;
      =     "DB_ACHSE13".A_SGselect1;
      =     "DB_ACHSE14".A_SGselect1;
NETWORK
TITLE =SG 1 -Auswahl Werkzeugwechsler / Magazin

      U     "DB_SPL".OI_SG_AUSW_34_MAGAX;
      =     "DB_ACHSE7".A_SGselect1;
      =     "DB_ACHSE13".A_SGselect1;
      =     "DB_ACHSE14".A_SGselect1;
NETWORK
TITLE =Spindel aktuelle Getriebstufe kopieren --> Anw. Meisel

      U     "DB_ACHSE6_SPINDEL".A_ActGearA;
      =     "DB_ACHSE6_SPINDEL".A_Transmiss0;

      U     "DB_ACHSE6_SPINDEL".A_ActGearB;
      =     "DB_ACHSE6_SPINDEL".A_Transmiss1;

      U     "DB_ACHSE6_SPINDEL".A_ActGearC;
      =     "DB_ACHSE6_SPINDEL".A_Transmiss2;


NETWORK
TITLE =PLC-->NC: PS: SBH Anforderung durch Anwahl Entriegeln
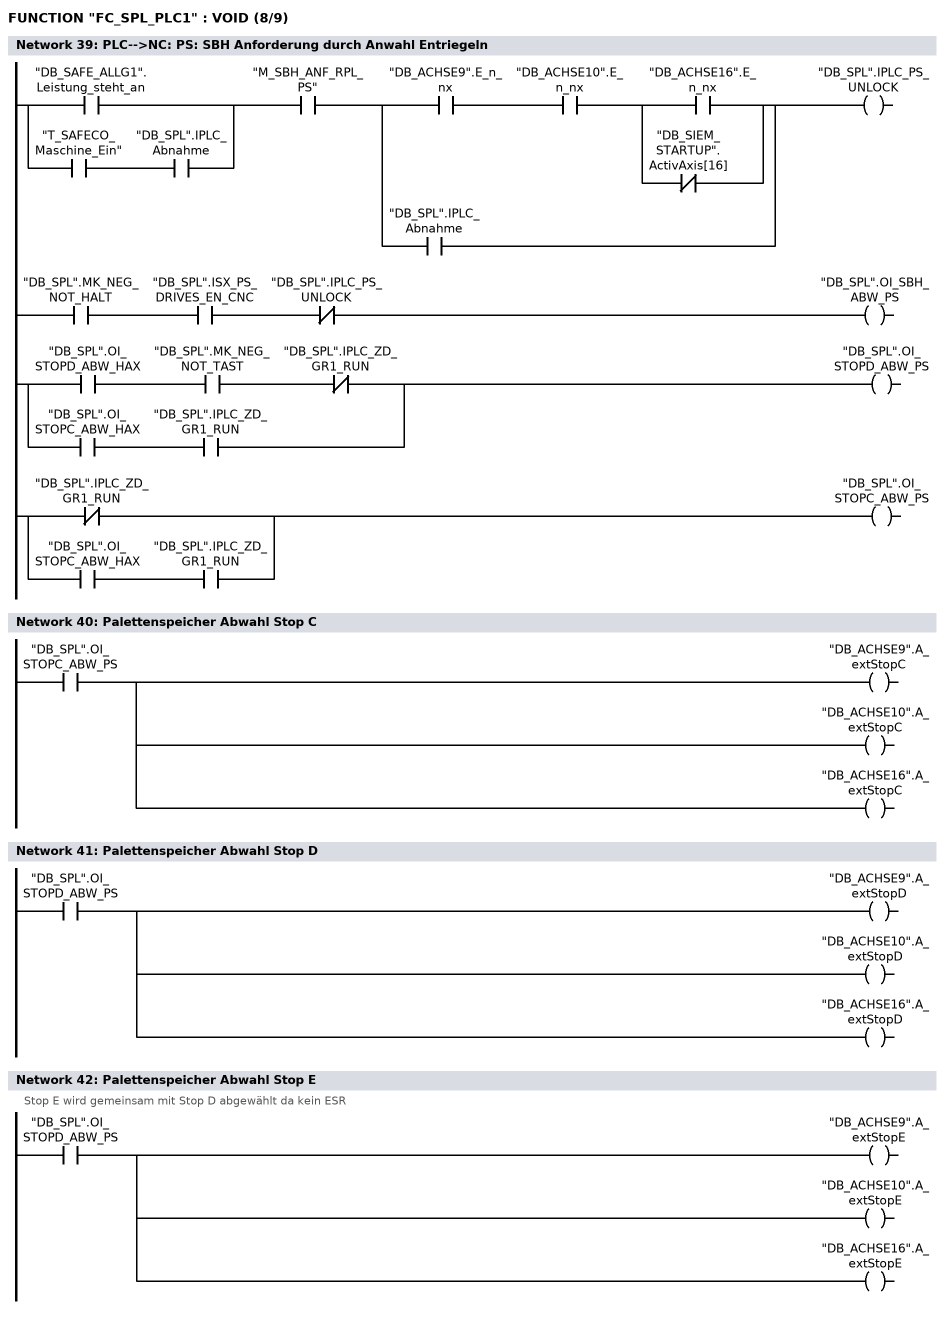

      U(    ;
      O     "DB_SAFE_ALLG1".Leistung_steht_an;
      O     ;
      U     "T_SAFECO_Maschine_Ein";
      U     "DB_SPL".IPLC_Abnahme;
      )     ;
      U     "M_SBH_ANF_RPL_PS";
      U(    ;
      U     "DB_ACHSE9".E_n_nx;
      U     "DB_ACHSE10".E_n_nx;
      U(    ;
      O     "DB_ACHSE16".E_n_nx;
      ON    "DB_SIEM_STARTUP".ActivAxis[16];
      )     ;
      O     "DB_SPL".IPLC_Abnahme;
      )     ;
      =     "DB_SPL".IPLC_PS_UNLOCK;

// SBH-Abwahl-
      U     "DB_SPL".MK_NEG_NOT_HALT;
      U     "DB_SPL".ISX_PS_DRIVES_EN_CNC;
      UN    "DB_SPL".IPLC_PS_UNLOCK;
      =     "DB_SPL".OI_SBH_ABW_PS;


//--- Externer Stopp D- Abwahl : Rundspeicherachse

      O(    ;
      U     "DB_SPL".OI_STOPD_ABW_HAX;
      U     "DB_SPL".MK_NEG_NOT_TAST;
      UN    "DB_SPL".IPLC_ZD_GR1_RUN;
      )     ;
      O(    ;
      U     "DB_SPL".OI_STOPC_ABW_HAX;
      U     "DB_SPL".IPLC_ZD_GR1_RUN;
      )     ;
      =     "DB_SPL".OI_STOPD_ABW_PS;

			//--- Externer Stopp C - Abwahl : Rundspeicherachse

      UN    "DB_SPL".IPLC_ZD_GR1_RUN;
      O(    ;
      U     "DB_SPL".OI_STOPC_ABW_HAX;
      U     "DB_SPL".IPLC_ZD_GR1_RUN;
      )     ;
      =     "DB_SPL".OI_STOPC_ABW_PS;

NETWORK
TITLE =Palettenspeicher Abwahl Stop C

      U     "DB_SPL".OI_STOPC_ABW_PS;
      =     "DB_ACHSE9".A_extStopC;
      =     "DB_ACHSE10".A_extStopC;
      =     "DB_ACHSE16".A_extStopC;

NETWORK
TITLE =Palettenspeicher Abwahl Stop D

      U     "DB_SPL".OI_STOPD_ABW_PS;
      =     "DB_ACHSE9".A_extStopD;
      =     "DB_ACHSE10".A_extStopD;
      =     "DB_ACHSE16".A_extStopD;

NETWORK
TITLE =Palettenspeicher Abwahl Stop E
//Stop E wird gemeinsam mit Stop D abgewählt da kein ESR
      U     "DB_SPL".OI_STOPD_ABW_PS;
      =     "DB_ACHSE9".A_extStopE;
      =     "DB_ACHSE10".A_extStopE;
      =     "DB_ACHSE16".A_extStopE;

NETWORK
TITLE =Abwahl SBH Palettenspeicher
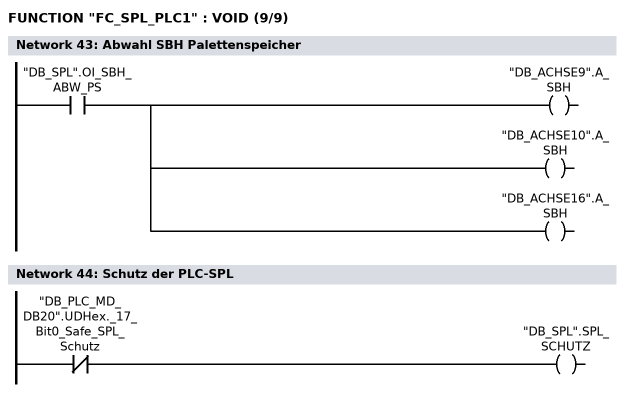

      U     "DB_SPL".OI_SBH_ABW_PS;
      =     "DB_ACHSE9".A_SBH;
      =     "DB_ACHSE10".A_SBH;
      =     "DB_ACHSE16".A_SBH;

NETWORK
TITLE =Schutz der PLC-SPL

      UN    "DB_PLC_MD_DB20".UDHex._17_Bit0_Safe_SPL_Schutz;
      =     "DB_SPL".SPL_SCHUTZ;
END_FUNCTION

